(* CODESYS project Elevator.project

Project tree, tasks and I/O mapping:
  Device : Elmo Platinum Maestro, Elmo Motion Control, version 1.0.0.2
    application Application
      libraries: Standard, * (System); VisuDialogs, * (System)
      task MainTask (cyclic, interval t#20ms, priority 1) calls nothing
      task VISU_TASK (cyclic, interval 100 ms, priority 31) calls VisuElems.Visu_Prg, PLC_PRG
      visualisation Visualization
      visualisation Elavator
      function block FB_Elevator [ST]: M_Enter, M_OpenDoor, M_Exit, M_Move, M_DisplayDirection, M_CloseDoor, M_DisplayNextFloor, M_DisplayNowFloor, M_FloorBtnClick, M_DisplayDoorState, M_IsMoving, M_IsAtFloor, M_StopMoving, M_IsDoorOpen
      data type st_Elevator
      interface ITF_Action: M_OpenDoor, M_CloseDoor, M_Move, M_FloorBtnClick
      function block FB_PassenEle [ST]
      function block FB_FreightEle [ST]: M_Move, M_Enter, M_Exit, M_Apperance
      interface ITF_Display: M_DisplayNowFloor, M_DisplayNextFloor, M_DisplayDirection, M_DisplayDoorState
      interface ITF_Counting: M_Enter, M_Exit
      visualisation OutsideEle
      visualisation FreightElavator
      function block Floor [ST]: M_GetPassengerCount, M_SetPassengerCount, M_AddPassenger, M_DelPassenger
    Maestro : Maestro, Elmo, version 1.0.0.2
  text list GlobalTextList
*)

// Device/Application/st_Elevator
TYPE st_Elevator :
STRUCT
	xKey  : ARRAY [1..5] OF BOOL;
	iFloor: BOOL;
	xEnter : BOOL;
	xExit : BOOL;
	EleState : STRING;
	ODoor :  BOOL;
	CDoor :  BOOL;
	iWay :  STRING;
	iNextFloor : STRING;
	iNowFloor : STRING;
	//ix_Start : BOOL;
END_STRUCT
END_TYPE

// Device/Application/FB_Elevator
FUNCTION_BLOCK FB_Elevator IMPLEMENTS ITF_Action,ITF_Display,ITF_Counting
VAR_INPUT
	ix_Start  : BOOL;
	xKey  : ARRAY [0..5] OF BOOL;
	ODoor : BOOL;
	CDoor : BOOL;
	Enter : BOOL;
	iPos : INT;
	iWaitingCounter : INT;
END_VAR
VAR_OUTPUT
	
END_VAR
VAR
	
	FloorNow  : INT :=1;
	TargetFloor  :INT :=1;
	direction : INT := 0;
	doorstate : BOOL := FALSE;  
	DoorDisplay : STRING;
	Light: BOOL := FALSE; 
	
	iMove : INT;
	
	
	passengerCount : INT := 0;
    maxCapacity    : INT := 3;
	StrDir : STRING;
	count: UINT;
	Speed: INT := 1;
	
	iKeyClicked : INT;
	up : BOOL;
	down: BOOL;
	
	currentFloor: BOOL;
	xEnter : BOOL;
	xExit : BOOL;
	EleState : STRING;
	//ODoor :  BOOL;
	//CDoor :  BOOL;
	iWay :  STRING;
	iNextFloor : STRING;
	iNowFloor : STRING;
	
	os_Status : STRING;
	
	xDoorFullyOpen : BOOL;
	fbAutoCloseTimer : TON; 
	tDoorOpenDwellTime : TIME := T#5S;
	bAutoCloseTriggered : BOOL;
	
	bIsMoving : BOOL := FALSE;
	
	
	iMaxWaitingTime : INT := 300;
END_VAR
VAR CONSTANT
END_VAR

fbAutoCloseTimer.IN := xDoorFullyOpen;
fbAutoCloseTimer.PT := tDoorOpenDwellTime;
fbAutoCloseTimer ();

IF fbAutoCloseTimer.Q AND (DoorState = FALSE) AND NOT bAutoCloseTriggered THEN
	THIS^.M_CloseDoor(); 
	bAutoCloseTriggered := TRUE;
END_IF

METHOD M_Enter: BOOL
VAR_INPUT	
	count: INT;
END_VAR
IF passengerCount + count <= maxCapacity THEN
	passengerCount := passengerCount + count;
	M_Enter := TRUE; 
ELSE
	M_Enter := FALSE; 
END_IF;
END_METHOD

METHOD M_OpenDoor : BOOL
VAR_INPUT
END_VAR
doorstate:= TRUE;
END_METHOD

METHOD M_Exit : BOOL
VAR_INPUT
	count: INT;
END_VAR
IF passengerCount - count >= 0 THEN
	passengerCount := passengerCount - count;
	M_Exit := TRUE;
ELSE
	passengerCount := 0;
	M_Exit := TRUE;
END_IF;
END_METHOD

METHOD M_Move : BOOL
VAR_INPUT
	 floor : INT;
END_VAR
IF (floor < -1) OR (floor > 5) THEN
        M_Move := FALSE; 
		 
ELSE
     TargetFloor := floor;
IF targetFloor > FloorNow  THEN
        direction := 1;
		Light := TRUE;
		
    ELSIF targetFloor < FloorNow THEN
        direction := -1;
    ELSE
        direction := 0;
		Light := FALSE;
    END_IF;   
END_IF;	
 FloorNow := targetFloor;
END_METHOD

METHOD M_DisplayDirection : STRING
VAR_INPUT
END_VAR
CASE direction OF
	1: StrDir := 'Going Up';
   -1: StrDir := 'Going Down';
ELSE
	StrDir := 'Pending';
END_CASE;
M_DisplayDirection := StrDir;
END_METHOD

METHOD M_CloseDoor : BOOL
VAR_INPUT
END_VAR
doorstate:= FALSE;
END_METHOD

METHOD M_DisplayNextFloor : STRING
VAR_INPUT
END_VAR
IF TargetFloor > 0 AND TargetFloor < 6 THEN
	M_DisplayNextFloor :=INT_TO_STRING(TargetFloor);
ELSIF TargetFloor = 0 THEN
	M_DisplayNextFloor :='B1';
ELSE 
	M_DisplayNextFloor := 'Error';
END_IF
END_METHOD

METHOD M_DisplayNowFloor : STRING
VAR_INPUT
END_VAR
IF FloorNow > 0 AND FloorNow < 6 THEN
	M_DisplayNowFloor :=INT_TO_STRING(FloorNow);
ELSIF TargetFloor = 0 THEN
	M_DisplayNowFloor :='B1';
ELSE 
	M_DisplayNowFloor := 'Error';
END_IF
END_METHOD

METHOD M_FloorBtnClick : BOOL
VAR_INPUT
	xNumber  : BOOL;
END_VAR

VAR
	i: INT;
END_VAR
IF xKey[1] THEN
	iKeyClicked := 1;
ELSIF xKey[2] THEN
	iKeyClicked := 2;
ELSIF xKey[3] THEN
	iKeyClicked := 3;	
ELSIF xKey[4] THEN
	iKeyClicked := 4;	
ELSIF xKey[5] THEN
	iKeyClicked := 5;	
END_IF


IF iKeyClicked < 1 OR iKeyClicked > 5 THEN
	M_FloorBtnClick := FALSE;
	RETURN;
END_IF

FOR i := 1 TO 5 DO
	IF ix_Start = FALSE AND xKey[i] = FALSE THEN
		ix_Start := TRUE;
		TargetFloor := iKeyClicked;
	END_IF

END_FOR

M_FloorBtnClick := TRUE;
END_METHOD

METHOD M_DisplayDoorState : STRING
VAR_INPUT
END_VAR
IF doorstate THEN
	DoorDisplay := 'Open';
ELSE
	DoorDisplay := 'Close';
END_IF;
M_DisplayDoorState :=DoorDisplay;
END_METHOD

METHOD M_IsMoving : BOOL
VAR_INPUT
END_VAR
M_IsMoving := bIsMoving;;
END_METHOD

METHOD M_IsAtFloor : BOOL
VAR_INPUT
	floorCoordinates : ARRAY[1..5] OF INT;
END_VAR
VAR
	i : INT;
END_VAR
VAR CONSTANT
	EPS : INT := 1;
END_VAR
FOR i := 1 TO 5 BY 1 DO
	IF ABS(iPos - floorCoordinates[i]) <= EPS THEN
		M_IsAtFloor := TRUE;
		RETURN;
	END_IF
END_FOR
M_IsAtFloor := FALSE;
END_METHOD

METHOD M_StopMoving
VAR_INPUT
END_VAR
iWaitingCounter := 0;
bIsMoving := FALSE;
END_METHOD

METHOD M_IsDoorOpen : BOOL
VAR_INPUT
END_VAR
M_IsDoorOpen := doorstate;
END_METHOD

END_FUNCTION_BLOCK

// Device/Application/ITF_Action
INTERFACE ITF_Action

METHOD M_OpenDoor : BOOL
VAR_INPUT
END_VAR
END_METHOD

METHOD M_CloseDoor : BOOL
VAR_INPUT
END_VAR
END_METHOD

METHOD M_Move : BOOL
VAR_INPUT
	floor : INT;
END_VAR
END_METHOD

METHOD M_FloorBtnClick : BOOL
VAR_INPUT
	xNumber  : BOOL;
END_VAR
END_METHOD

END_INTERFACE

// Device/Application/Floor
FUNCTION_BLOCK Floor
VAR
	passengerCount : INT;
END_VAR

METHOD M_GetPassengerCount : INT
VAR_INPUT
END_VAR
M_GetPassengerCount := passengerCount;
END_METHOD

METHOD M_SetPassengerCount
VAR_INPUT
	count : INT;
END_VAR
passengerCount := count;
END_METHOD

METHOD M_AddPassenger : BOOL
VAR_INPUT
END_VAR
passengerCount := passengerCount + 1;
END_METHOD

METHOD M_DelPassenger : BOOL
VAR_INPUT
END_VAR
IF passengerCount >= 1 THEN
	passengerCount := passengerCount - 1;
END_IF
END_METHOD

END_FUNCTION_BLOCK

// Device/Application/ITF_Display
INTERFACE ITF_Display

METHOD M_DisplayNowFloor : STRING
VAR_INPUT
END_VAR
END_METHOD

METHOD M_DisplayNextFloor : STRING
VAR_INPUT
END_VAR
END_METHOD

METHOD M_DisplayDirection : STRING
VAR_INPUT
END_VAR
END_METHOD

METHOD M_DisplayDoorState : STRING
VAR_INPUT
END_VAR
END_METHOD

END_INTERFACE

// Device/Application/ITF_Counting
INTERFACE ITF_Counting

METHOD M_Enter : BOOL
VAR_INPUT
	count : INT;
END_VAR
END_METHOD

METHOD M_Exit : BOOL
VAR_INPUT
	count: INT;
END_VAR
END_METHOD

END_INTERFACE

// Device/Application/FB_PassenEle
FUNCTION_BLOCK FB_PassenEle EXTENDS FB_Elevator 
VAR_INPUT
END_VAR
VAR_OUTPUT
END_VAR
VAR
	
END_VAR

END_FUNCTION_BLOCK

// Device/Application/FB_FreightEle
FUNCTION_BLOCK FB_FreightEle EXTENDS FB_PassenEle
VAR_INPUT
	
END_VAR
VAR_OUTPUT
END_VAR
VAR
	FreightCount : INT := 0;
	Capacitymax    : INT := 5;
	//count: UINT;
	iState : INT;
	
END_VAR

SUPER^();

METHOD M_Move : BOOL
VAR_INPUT
	 floor : INT;
END_VAR

VAR
	
END_VAR
IF (floor < -1) OR (floor > 5) THEN
        M_Move := FALSE; 
		 
ELSE
     TargetFloor := floor;
IF targetFloor > FloorNow  THEN
        direction := 1;
		Light := TRUE;
		
    ELSIF targetFloor < FloorNow THEN
        direction := -1;
    ELSE
        direction := 0;
		Light := FALSE;
    END_IF;   
END_IF;	
 FloorNow := targetFloor;
END_METHOD

METHOD M_Enter : BOOL
VAR_INPUT
	count : INT;
END_VAR
IF FreightCount + count <= Capacitymax THEN
        FreightCount := FreightCount + count;
        M_Enter := TRUE;
    ELSE
        M_Enter := FALSE;
    END_IF;
END_METHOD

METHOD M_Exit : BOOL
VAR_INPUT
	count: INT;
END_VAR
IF passengerCount - count >= 0 THEN
        passengerCount := passengerCount - count;
        M_Exit := TRUE;
    ELSE
        passengerCount := 0;
        M_Exit := TRUE;
    END_IF;
END_METHOD

METHOD M_Apperance
VAR_INPUT
END_VAR
END_METHOD

END_FUNCTION_BLOCK

// Device/Application/Visualization
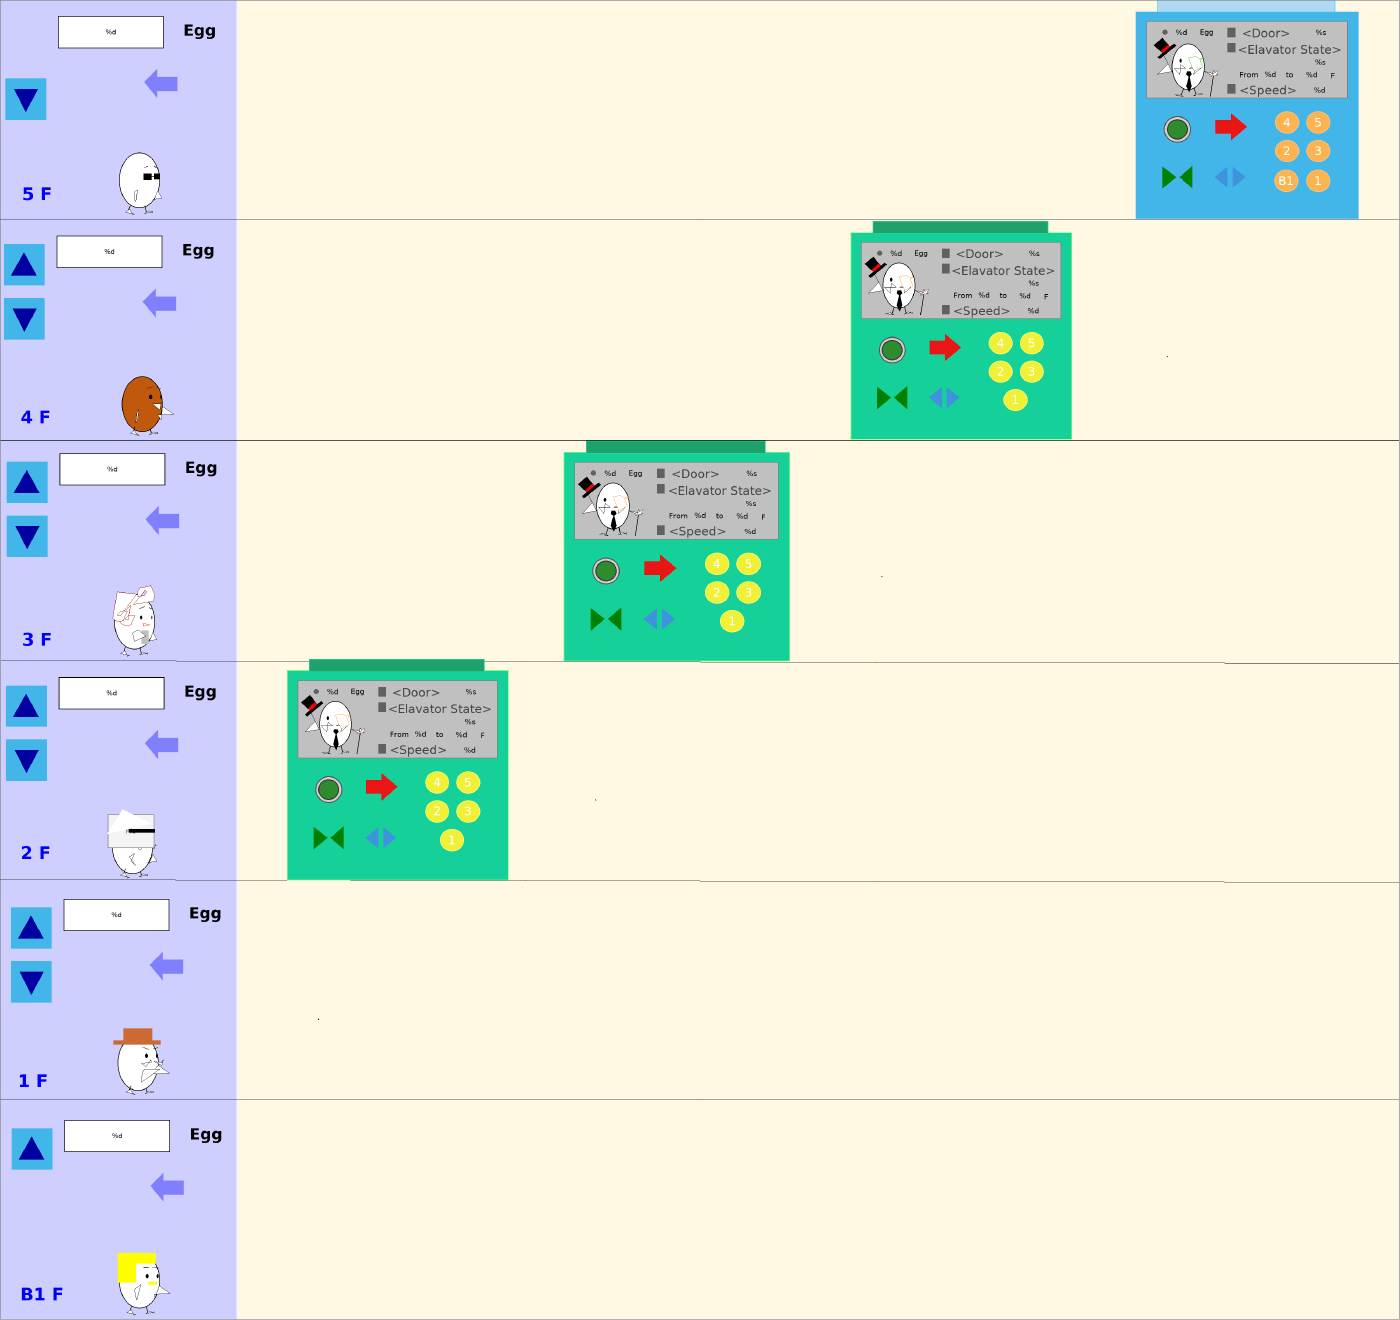
VISUALIZATION Visualization  // 2000x1887
    Rectangle (339,0 1661x1886)
    Rectangle (-4,0 342x1887)
    Line (2,944) (1999,948)
    Line (1,629) (1999,629)
    Line (1,313) (2003,314)
    Line (-2,1571) (1998,1572)
    Frame (805,630 323x316)
        shows Elavator(fbElevatorVisu := PLC_PRG.fbElevator[2])
        p2738717112: PLC_PRG.fbElevator[2].iMove
    Frame (1215,316 316x313)
        shows Elavator(fbElevatorVisu := PLC_PRG.fbElevator[3])
        p2738717112: PLC_PRG.fbElevator[3].iMove
    Line (1,1257) (1998,1261)
    Group (162,1470 80x95)
        Line (48,91) (46,82)
        Polygon (45,93) (51,89) (57,92) (57,90)
        Ellipse (6,10 58x79)
        Polygon (55,63) (57,65) (80,64) (64,53)
        Polygon (44,58) (41,64) (40,77) (66,58)
        Line (22,90) (25,82)
        Polygon (18,91) (24,87) (28,95) (31,94)
        Rectangle (0,17 67x6)
        Rectangle (14,0 41x17)
        Polygon (58,47) (69,53) (71,45) (69,49)
        Polygon (40,50) (46,55) (53,45) (54,48)
        Ellipse (45,36 4x6)
        Ellipse (61,36 2x6)
        Line (50,30) (42,27)
        Line (57,29) (63,27)
    Group (153,1157 71x98)
        Line (49,94) (47,85)
        Polygon (46,96) (52,92) (58,95) (58,93)
        Ellipse (7,13 58x79)
        Polygon (60,77) (58,76) (71,74) (65,64)
        Polygon (39,63) (31,68) (41,80) (34,74)
        Line (23,93) (26,85)
        Polygon (19,94) (25,90) (29,98) (32,97)
        Polygon (59,50) (67,56) (69,50) (70,52)
        Polygon (42,54) (47,58) (54,48) (55,51)
        Ellipse (46,39 4x6)
        Ellipse (62,39 2x6)
        Line (51,33) (44,35)
        Line (58,32) (63,35)
        Pie (1,7 66x48)
        Rectangle (31,28 37x5)
        Polygon (63,20) (22,0) (0,35) (0,35)
    Group (161,837 63x101)
        Ellipse (2,12 58x79)
        Line (41,97) (39,88)
        Polygon (38,99) (44,95) (50,98) (50,96)
        Polygon (52,80) (50,79) (63,77) (57,67)
        Line (15,96) (18,88)
        Polygon (11,97) (17,93) (21,101) (24,100)
        Ellipse (39,43 3x5)
        Ellipse (55,43 1x5)
        Line (45,30) (38,33)
        Line (52,31) (55,33)
        Polygon (43,54) (44,58) (53,56) (49,55)
        RoundedRectangle (41,64 10x19)
        Polygon (29,27) (58,22) (60,12) (58,9) (54,0) (45,2) (39,3) (35,9) (36,16) (45,14) (48,9) (46,6) (42,12)
        Polygon (25,28) (9,48) (11,53) (15,56) (19,57) (26,56) (28,50) (32,43) (27,42) (22,43) (17,48) (17,48) (22,49)
        Polygon (34,12) (6,9) (0,47) (4,50) (8,51) (15,50) (17,44) (21,37) (16,36) (11,37) (6,42) (6,42) (11,43)
        Polygon (36,63) (28,68) (31,80) (47,72)
    Group (170,218 61x89)
        Ellipse (0,0 58x79)
        Line (39,85) (37,76)
        Polygon (36,87) (42,83) (48,86) (48,84)
        Polygon (50,68) (48,67) (61,65) (55,55)
        Line (13,84) (16,76)
        Polygon (9,85) (15,81) (19,89) (22,88)
        Ellipse (37,31 3x5)
        Ellipse (53,31 1x5)
        Line (41,20) (36,21)
        Line (50,19) (53,21)
        RoundedRectangle (35,30 11x9)
        Polygon (26,53) (22,56) (22,68) (24,70)
        RoundedRectangle (50,30 8x8)
        Line (50,34) (46,34)
    Group (174,538 74x85)
        Line (42,81) (40,72)
        Polygon (39,83) (45,79) (51,82) (51,80)
        Ellipse (0,0 58x79)
        Polygon (56,62) (51,55) (74,54) (58,43)
        Polygon (24,47) (21,53) (20,66) (22,62)
        Line (16,80) (19,72)
        Polygon (12,81) (18,77) (22,85) (25,84)
        Polygon (44,39) (54,48) (56,37) (57,39)
        Ellipse (39,26 4x6)
        Ellipse (55,26 2x6)
        Line (43,15) (36,17)
        Line (50,15) (55,17)
    Group (168,1791 75x89)
        Line (43,85) (41,76)
        Polygon (40,87) (46,83) (52,86) (52,84)
        Ellipse (2,0 58x79)
        Polygon (53,65) (52,59) (75,58) (59,47)
        Polygon (24,52) (25,58) (27,67) (33,45)
        Line (17,84) (20,76)
        Polygon (13,85) (19,81) (23,89) (26,88)
        Rectangle (0,11 26x31)
        Rectangle (0,0 54x15)
        Ellipse (40,30 4x6)
        Ellipse (56,30 2x6)
        Line (44,21) (37,21)
        Line (50,20) (58,21)
        Rectangle (44,41 12x4)
    Rectangle (1924,-301 135x76)
    Rectangle (17,1814 86x72), "B1 F"
    Rectangle (4,1509 86x72), "1 F"
    Rectangle (8,1183 86x72), "2 F"
    Rectangle (10,878 86x72), "3 F"
    Rectangle (8,560 86x72), "4 F"
    Rectangle (6,241 86x72), "5 F"
    Frame (15,1273 319x161)
        shows OutsideEle()
    Frame (8,956 319x161)
        shows OutsideEle()
    Frame (16,1589 319x161)
        shows OutsideEle()
    Frame (9,636 319x161)
        shows OutsideEle()
    Frame (5,325 319x161)
        shows OutsideEle()
    Frame (7,11 319x161)
        shows OutsideEle()
    Rectangle (5,27 66x71)
    Rectangle (15,1688 66x71)
    Frame (410,942 316x317)
        shows Elavator(fbElevatorVisu := PLC_PRG.fbElevator[1])
    Frame (1622,0 319x314)
        shows FreightElavator(fbFreightVisu := PLC_PRG.FreightEle)
END_VISUALIZATION

// Device/Application/Elavator
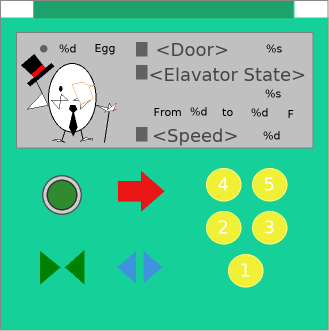
VISUALIZATION Elavator  // 329x331
VAR_IN_OUT
	fbElevatorVisu  : fb_Elevator;
END_VAR
    Polyline (46,537) (47,538)
    RoundedRectangle (0,17 329x313)
    RoundedRectangle (16,32 297x116)
    Ellipse (252,168 35x33), "5"
        tap fbElevatorVisu.xKey[5]
        OnMouseClick: execute {  }
    Ellipse (252,211 35x33), "3"
        tap fbElevatorVisu.xKey[3]
        OnMouseClick: execute {  }
    Ellipse (206,168 35x33), "4"
        tap fbElevatorVisu.xKey[4]
        OnMouseClick: execute {  }
    Ellipse (206,211 35x33), "2"
        tap fbElevatorVisu.xKey[2]
        OnMouseClick: execute {  }
    Ellipse (228,254 35x33), "1"
        tap fbElevatorVisu.xKey[1]
        OnMouseClick: execute {  }
    Lamp1 (39,170 46x50), variable: fbElevatorVisu.Light, style: Lamp-Lamp1-Green
    Polygon (141,171) (164,191) (141,211) (141,201) (118,201) (118,181) (141,181)
        tap fbElevatorVisu.Enter
        OnMouseClick: execute { fbElevatorVisu.M_Enter(1); }
    Rectangle (37,39 62x20), "%d", text variable: fbElevatorVisu.passengerCount
    Rectangle (136,42 11x14)
    Label (108,37 169x26), "<Door>"
    Rectangle (237,40 74x18), "%s", text variable: fbElevatorVisu.DoorDisplay
    Rectangle (223,104 74x18), "%d", text variable: fbElevatorVisu.TargetFloor
    Rectangle (136,65 11x14)
    Label (143,62 169x26), "<Elavator State>"
    Rectangle (236,85 74x18), "%s", text variable: fbElevatorVisu.M_DisplayDirection()
    Label (277,106 28x17), "F"
    Label (85,30 40x37), "Egg"
    Ellipse (40,45 7x7)
    Rectangle (33,0 261x19)
    Group (21,54 95x88)
        Ellipse (27,9 48x69)
        Line (41,86) (44,77)
        Line (62,85) (60,76)
        Ellipse (38,32 3x5)
        Ellipse (56,32 3x5)
        Polygon (75,51) (86,57) (88,49) (92,55)
        Polygon (69,46) (59,55) (61,42) (52,46)
        Polygon (30,46) (38,55) (40,40) (47,46)
        Polygon (15,27) (21,39) (6,55) (27,51)
        Polygon (59,87) (65,83) (71,86) (71,84)
        Line (88,55) (83,88)
        Polygon (83,58) (95,49) (92,57) (95,55)
        Polygon (31,86) (39,85) (39,86) (44,88)
        Polygon (9,32) (33,12) (30,9) (24,14) (13,0) (0,11) (13,23) (6,29)
        Polygon (13,24) (24,14) (21,10) (10,20) (13,23)
        Polygon (68,33) (72,44) (60,50) (55,41) (51,30) (62,28) (67,31) (75,31)
        Group (48,51 4x23)
            Polygon (1,0) (6,0) (8,4) (4,8) (0,4)
            Polygon (4,5) (8,22) (4,31) (0,22)
    Rectangle (162,103 74x18), "%d", text variable: fbElevatorVisu.FloorNow
        OnMouseClick: write the text variable via Default
    Label (214,104 27x17), "to"
    Label (153,104 29x17), "From"
    Rectangle (136,127 11x14)
    Label (111,123 169x26), "<Speed>"
    Rectangle (235,127 74x18), "%d", text variable: fbElevatorVisu.Speed
        OnMouseClick: write the text variable via Default
    Polygon (137,250) (142,250) (162,267) (142,284) (137,284) (137,284) (117,267)
        tap fbElevatorVisu.ODoor
    Rectangle (136,240 7x50)
    Polygon (84,250) (84,284) (65,267) (60,267) (40,284) (40,251) (60,267) (65,267)
        tap fbElevatorVisu.CDoor
    Rectangle (61,241 3x50)
END_VISUALIZATION

// Device/Application/OutsideEle
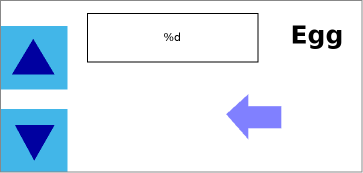
VISUALIZATION OutsideEle  // 363x173
VAR_IN_OUT
	fbEleOutsideVisu  : fb_Elevator;
END_VAR
    RoundedRectangle (1,26 66x63)
        toggle fbEleOutsideVisu.up
    Polygon (33,39) (12,74) (54,74)
    RoundedRectangle (1,109 66x63)
        toggle fbEleOutsideVisu.down
    Polygon (15,125) (34,160) (54,125)
    Rectangle (87,13 171x49), "%d"
    Label (292,13 50x43), "Egg"
    Polygon (226,114) (248,94) (248,106) (281,106) (281,128) (248,128) (248,139), text variable: fbElevatorVisu.Speed
        tap fbElevatorVisu.xExit
END_VISUALIZATION

// Device/Application/FreightElavator
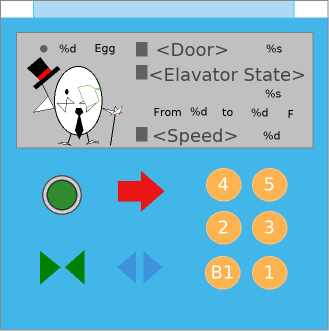
VISUALIZATION FreightElavator  // 329x331
VAR_IN_OUT
	fbFreightVisu  : FB_FreightEle;
END_VAR
    Polyline (46,537) (47,538)
    RoundedRectangle (0,17 329x313)
    RoundedRectangle (16,32 297x116)
    Ellipse (252,168 35x33), "5"
        tap fbFreightVisu.xKey[5]
        OnMouseClick: execute {  }
    Ellipse (252,211 35x33), "3"
        tap fbFreightVisu.xKey[3]
        OnMouseClick: execute {  }
    Ellipse (206,168 35x33), "4"
        tap fbFreightVisu.xKey[4]
        OnMouseClick: execute {  }
    Ellipse (206,211 35x33), "2"
        tap fbFreightVisu.xKey[2]
        OnMouseClick: execute {  }
    Ellipse (252,256 35x33), "1"
        tap fbFreightVisu.xKey[1]
        OnMouseClick: execute {  }
    Lamp1 (39,170 46x50), variable: fbElevatorVisu.Light, style: Lamp-Lamp1-Green
    Polygon (141,171) (164,191) (141,211) (141,201) (118,201) (118,181) (141,181)
        tap fbElevatorVisu.Enter
        OnMouseClick: execute { fbElevatorVisu.M_Enter(1); }
    Rectangle (37,39 62x20), "%d", text variable: fbElevatorVisu.passengerCount
    Rectangle (136,42 11x14)
    Label (108,37 169x26), "<Door>"
    Rectangle (237,40 74x18), "%s", text variable: fbElevatorVisu.DoorDisplay
    Rectangle (223,104 74x18), "%d", text variable: fbElevatorVisu.TargetFloor
    Rectangle (136,65 11x14)
    Label (143,62 169x26), "<Elavator State>"
    Rectangle (236,85 74x18), "%s", text variable: fbElevatorVisu.M_DisplayDirection()
    Label (277,106 28x17), "F"
    Label (85,30 40x37), "Egg"
    Ellipse (40,45 7x7)
    Rectangle (33,-1 261x19)
    Group (27,57 95x88)
        Ellipse (27,9 48x69)
        Line (41,86) (44,77)
        Line (62,85) (60,76)
        Ellipse (38,32 3x5)
        Ellipse (56,32 3x5)
        Polygon (75,51) (86,57) (88,49) (92,55)
        Polygon (69,46) (59,55) (61,42) (52,46)
        Polygon (30,46) (38,55) (40,40) (47,46)
        Polygon (15,27) (21,39) (6,55) (27,51)
        Polygon (59,87) (65,83) (71,86) (71,84)
        Line (88,55) (83,88)
        Polygon (83,58) (95,49) (92,57) (95,55)
        Polygon (31,86) (39,85) (39,86) (44,88)
        Polygon (9,32) (33,12) (30,9) (24,14) (13,0) (0,11) (13,23) (6,29)
        Polygon (13,24) (24,14) (21,10) (10,20) (13,23)
        Polygon (68,33) (72,44) (60,50) (55,41) (51,30) (62,28) (67,31) (75,31)
        Group (48,51 4x23)
            Polygon (1,0) (6,0) (8,4) (4,8) (0,4)
            Polygon (4,5) (8,22) (4,31) (0,22)
    Rectangle (162,103 74x18), "%d", text variable: fbElevatorVisu.FloorNow
        OnMouseClick: write the text variable via Default
    Label (214,104 27x17), "to"
    Label (153,104 29x17), "From"
    Rectangle (136,127 11x14)
    Label (111,123 169x26), "<Speed>"
    Rectangle (235,127 74x18), "%d", text variable: fbElevatorVisu.Speed
        OnMouseClick: write the text variable via Default
    Polygon (137,250) (142,250) (162,267) (142,284) (137,284) (137,284) (117,267)
        tap fbElevatorVisu.ODoor
    Rectangle (136,240 7x50)
    Polygon (84,250) (84,284) (65,267) (60,267) (40,284) (40,251) (60,267) (65,267)
        tap fbElevatorVisu.CDoor
    Rectangle (61,241 3x50)
    Ellipse (205,256 35x33), "B1"
        tap fbFreightVisu.xKey[0]
        OnMouseClick: execute {  }
END_VISUALIZATION
